// TIA Portal V19 export
FUNCTION_BLOCK "FB_SafeTest"   // FB500, F_LAD
{ S7_Optimized_Access := 'TRUE' }
VERSION : 0.1
// stored: AutoNumber false, IsIECCheckEnabled false, UDAEnableTagReadback false
   VAR_INPUT
      In1 : Bool;
   END_VAR
   VAR_OUTPUT
      Out1 : Bool;
   END_VAR
BEGIN

REGION Network 1
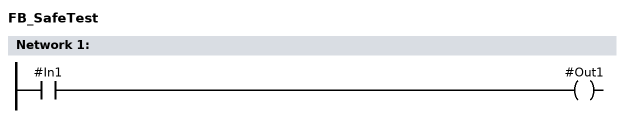
   RUNG wire#powerrail
      Contact( #In1 )
      Coil( #Out1 )
   END_RUNG
   // the same network as SCL:
   #Out1 := #In1;
END_REGION
END_FUNCTION_BLOCK
